INTERFACE I_Roof

METHOD Close : BOOL
VAR_INPUT
END_VAR
END_METHOD

METHOD Open : BOOL
VAR_INPUT
END_VAR
END_METHOD

METHOD Reset : BOOL
VAR_INPUT
END_VAR
END_METHOD

PROPERTY State : E_RoofState
GET
END_GET
END_PROPERTY

METHOD Stop : BOOL
VAR_INPUT
END_VAR
END_METHOD

END_INTERFACE

(* stored: Version 1.1.0.1, ProductVersion 3.1.4024.15
   Itf I_Roof: Id {fca33943-8ae8-4619-8aba-a9cc7530ccc6}
   Method Close: Id {2a5de17d-b0db-429d-b5d4-7bf8aa94c396}
   Method Open: Id {b0027d20-fad9-4b5e-89f3-643491aad030}
   Method Reset: Id {7ac4ab4b-1dc7-43d7-b41b-04995de189e4}
   Property State: Id {9d0e9ff5-3e4c-4491-9e51-534859a8107e}
   Get Get: Id {103715e1-874b-4449-b6dc-3e7edf4fcdf8}
   Method Stop: Id {7c78fc7d-6196-46aa-bb88-07ed0ce90889} *)
